{attribute 'qualified_only'}
VAR_GLOBAL
	Actual_Velocity   AT%I*   :DINT  := 0;
	


	Control_word      AT%Q*   :UINT  := 0;
	int_val           AT%Q*   :INT   := 0;
	Target_Velocity   AT%Q*   :DINT  := 0;	
END_VAR

(* stored: Version 1.1.0.1, ProductVersion 3.1.4024.12
   GVL GVL: Id {e9d1865c-37ec-476b-802d-7bbf4ea05cea} *)
